Staubli VAL3: TestSuccionar.pjx

--- TestSuccionar.pjx ---
Parameters version=s7.11.2 stackSize=5000 millimeterUnit=true
Program file=start.pgx
Program file=stop.pgx
Data file=TestSuccionar.dtx

--- TestSuccionar.dtx ---
mdesc mNomSpeed
jointRx JApproach1 = {j1=-7.51952088935441, j2=-3.64589777611851, j3=61.4224022246856, j4=180.000005008956, j5=-122.22350312171, j6=-7.51951491293889}
jointRx jGetCinta
pointRx pApprBins = {x=391.677006562633, y=-12.0780346417013, z=88.9240734189491, rx=-179.999995158748, ry=2.22468368245291E-06, rz=-2.86880296299408E-07, fatherId=world[0]}
tool tToolSuccion = {z=110, fatherId=flange[0], ioLink=valve1}

--- start.pgx ---
program start()
begin
  movej(JApproach1,tToolSuccion, mNomSpeed)
  waitEndMove()
  movej(jGetCinta, tToolSuccion, mNomSpeed)
  waitEndMove()
  open(tToolSuccion)
  waitEndMove()
  movej(pApprBins, tToolSuccion, mNomSpeed)
  waitEndMove()
  close(tToolSuccion)
  waitEndMove()
end
